% RSLogix 500 project Semaphore.RSS, saved by version 8.30.00.16 %
PROJECT "UNTITLED"    % processor: Bul.1763 MicroLogix 1100 Series B %

PROGRAM FILES
  LAD 2   9 rungs

DATA FILES
  O0 OUTPUT  4 elements
  I1 INPUT  6 elements
  S2 STATUS  66 elements
  B3 BINARY  1 elements
  T4 TIMER  5 elements
  C5 COUNTER  1 elements
  R6 CONTROL  1 elements
  N7 INTEGER  1 elements
  F8 FLOAT  1 elements

LADDER 2
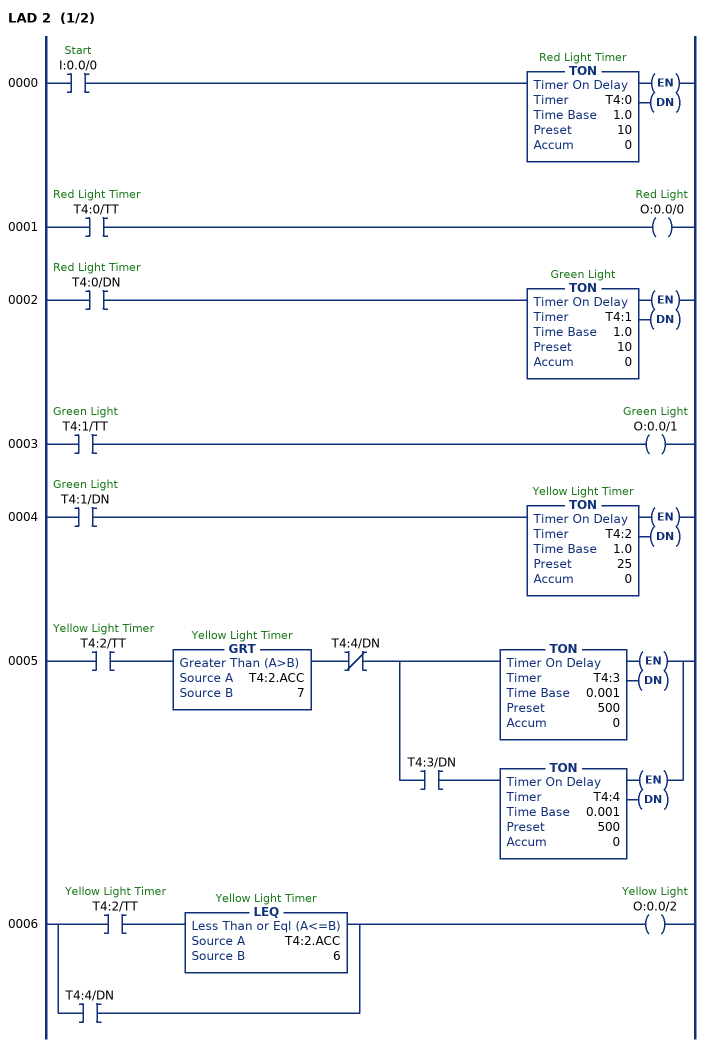
% Rung: 0 %
SOR XIC I:0.0/0 TON T4:0 1.0 10 0 EOR
%   I:0.0/0  "Start" %
%   T4:0  "Red Light Timer" %
% Rung: 1 %
SOR XIC T4:0/TT OTE O:0.0/0 EOR
%   T4:0  "Red Light Timer" %
%   O:0.0/0  "Red Light" %
% Rung: 2 %
SOR XIC T4:0/DN TON T4:1 1.0 10 0 EOR
%   T4:0  "Red Light Timer" %
%   T4:1  "Green Light" %
% Rung: 3 %
SOR XIC T4:1/TT OTE O:0.0/1 EOR
%   T4:1  "Green Light" %
%   O:0.0/1  "Green Light" %
% Rung: 4 %
SOR XIC T4:1/DN TON T4:2 1.0 25 0 EOR
%   T4:1  "Green Light" %
%   T4:2  "Yellow Light Timer" %
% Rung: 5 %
SOR XIC T4:2/TT GRT T4:2.ACC 7 XIO T4:4/DN BST TON T4:3 0.001 500 0 NXB XIC T4:3/DN TON T4:4 0.001 500 0 BND EOR
%   T4:2  "Yellow Light Timer" %
% Rung: 6 %
SOR BST XIC T4:2/TT LEQ T4:2.ACC 6 NXB XIC T4:4/DN BND OTE O:0.0/2 EOR
%   T4:2  "Yellow Light Timer" %
%   O:0.0/2  "Yellow Light" %

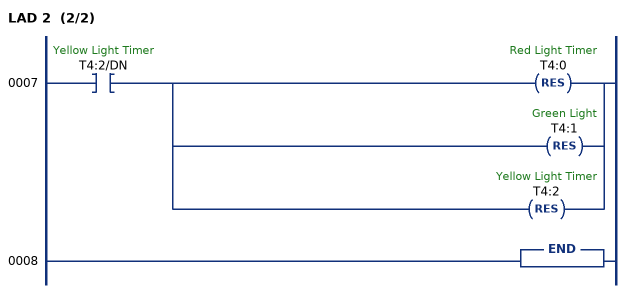
% Rung: 7 %
SOR XIC T4:2/DN BST RES T4:0 NXB RES T4:1 NXB RES T4:2 BND EOR
%   T4:2  "Yellow Light Timer" %
%   T4:0  "Red Light Timer" %
%   T4:1  "Green Light" %
% Rung: 8 %
SOR END EOR

DATA TABLE (non-zero values as saved)
DATA T4
% .PRE .ACC %
% T4:0 % 10 0
% T4:1 % 10 0
% T4:2 % 25 0
% T4:3 % 500 0
% T4:4 % 500 0
